KUKA KRL data list: InitProcessData.dat

&ACCESS RVO
&REL 83
&PARAM EDITMASK = *
&PARAM TEMPLATE = C:\KRC\Roboter\Template\vorgabe
&PARAM DISKPATH = KRC:\R1\Program\LeafProfiles
DEFDAT InitProcessData PUBLIC

   GLOBAL ENUM E_ProfileName FrameUpper,FrameHinge,FrameLock,FrameThreshold, LeafUpper,LeafBottom,LeafHinge,LeafLock

ENDDAT
